PROGRAM P5_00_MAIN
VAR

END_VAR

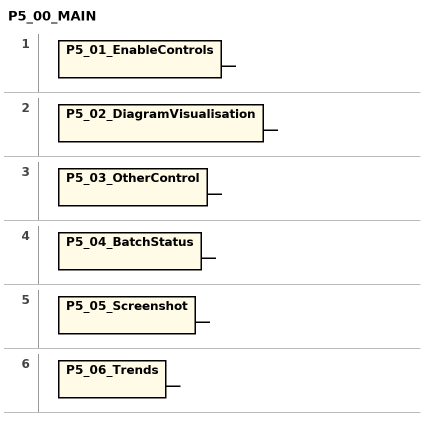
// NETWORK 1
P5_01_EnableControls();

// NETWORK 2
P5_02_DiagramVisualisation();

// NETWORK 3
P5_03_OtherControl();

// NETWORK 4
P5_04_BatchStatus();

// NETWORK 5
P5_05_Screenshot();

// NETWORK 6
P5_06_Trends();

END_PROGRAM

(* stored: Version 1.1.0.1
   POU P5_00_MAIN: Id {e5126a8f-d9ae-4302-9246-da3b2a0b21a1}, SpecialFunc None *)
